(* Logix 5000 project; controller PRU vendor 1 type 14 code 107 rev 20.13; software revision 20.01; part 10 of 17 *)
(* tags used below, declared in another part *)
   AFI : BOOL;
   CR0_CON1_HTR1_GON : BOOL;   // ZONE 1 (L1,L2,L3)
   CR1_CON2_HTR2_GON : BOOL;   // ZONE 2 (L1,L2,L3)
   CR2_CON3_HTR3_GON : BOOL;   // ZONE 3 (L1,L2,L3)
   CR3_CON4_HTR4_GON : BOOL;   // ZONE 4 (L1) ZONE 5 (L2) ZONE 6 (L3)
   CR4_CON5_HTR5_GON : BOOL;   // ZONE 7 (L1) ZONE 8 (L2) ZONE 9 (L3)
   CYCLE_ION_DELAY1_TON : TIMER;
   CYCLE_ION_DELAY2_TON : TIMER;
   CYCLE_ION_DELAY3_TON : TIMER;
   CYCLE_ION_DELAY4_TON : TIMER;
   HEATERS_CYCLE_ION : BOOL;   // Heaters are commanded on.
   HTR1_CV : REAL;
   HTR1_MAX_CV_LIMIT : REAL;
   HTR1_POWER_CMD : REAL;
   HTR2_CV : REAL;
   HTR2_MAX_CV_LIMIT : DINT;
   HTR2_POWER_CMD : REAL;
   HTR3_CV : REAL;
   HTR3_MAX_CV_LIMIT : REAL;
   HTR3_POWER_CMD : REAL;
   HTR4_CV : REAL;
   HTR4_MAX_CV_LIMIT : REAL;
   HTR4_POWER_CMD : REAL;
   HTR5_CV : REAL;
   HTR5_MAX_CV_LIMIT : REAL;
   HTR5_POWER_CMD : REAL;
   HTR6_CV : REAL;
   HTR6_MAX_CV_LIMIT : REAL;
   HTR6_POWER_CMD : REAL;
   HTR7_CV : REAL;
   HTR7_MAX_CV_LIMIT : REAL;
   HTR7_POWER_CMD : REAL;
   HTR8_CV : REAL;
   HTR8_MAX_CV_LIMIT : REAL;
   HTR8_POWER_CMD : REAL;
   HTR9_CV : REAL;
   HTR9_MAX_CV_LIMIT : REAL;
   HTR9_POWER_CMD : REAL;
   PID_1_MODE_LOCAL : BOOL;
   PID_2_MODE_LOCAL : BOOL;
   PID_3_MODE_LOCAL : BOOL;
   PID_4_MODE_LOCAL : BOOL;
   PID_5_MODE_LOCAL : BOOL;
   PID_6_MODE_LOCAL : BOOL;
   PID_7_MODE_LOCAL : BOOL;
   PID_8_MODE_LOCAL : BOOL;
   PID_9_MODE_LOCAL : BOOL;
   PID_ZONE_1 : PID;
   PID_ZONE_1_MANUAL_SETPOINT : REAL;
   PID_ZONE_1_SETPOINT : DINT;
   PID_ZONE_2 : PID;
   PID_ZONE_2_MANUAL_SETPOINT : REAL;
   PID_ZONE_2_SETPOINT : DINT;
   PID_ZONE_3 : PID;
   PID_ZONE_3_MANUAL_SETPOINT : REAL;
   PID_ZONE_3_SETPOINT : DINT;
   PID_ZONE_4 : PID;
   PID_ZONE_4_MANUAL_SETPOINT : REAL;
   PID_ZONE_4_SETPOINT : DINT;
   PID_ZONE_5 : PID;
   PID_ZONE_5_MANUAL_SETPOINT : REAL;
   PID_ZONE_5_SETPOINT : REAL;
   PID_ZONE_6 : PID;
   PID_ZONE_6_MANUAL_SETPOINT : REAL;
   PID_ZONE_6_SETPOINT : REAL;
   PID_ZONE_7 : PID;
   PID_ZONE_7_MANUAL_SETPOINT : REAL;
   PID_ZONE_7_SETPOINT : DINT;
   PID_ZONE_8 : PID;
   PID_ZONE_8_MANUAL_SETPOINT : REAL;
   PID_ZONE_8_SETPOINT : DINT;
   PID_ZONE_9 : PID;
   PID_ZONE_9_MANUAL_SETPOINT : REAL;
   PID_ZONE_9_SETPOINT : DINT;
   STANDBY_MODE_ION : BOOL;
   STANDBY_TEMPERATURE_SETPOINT : REAL;
   TEMPERATURE_SETPOINT_IS_RAMPING : BOOL;
   TEST_HTR1_CV_LIMIT : BOOL;
   TEST_HTR2_CV_LIMIT : BOOL;
   TEST_HTR3_CV_LIMIT : BOOL;
   TEST_HTR4_CV_LIMIT : BOOL;
   TEST_HTR5_CV_LIMIT : BOOL;
   TEST_HTR6_CV_LIMIT : BOOL;
   TEST_HTR7_CV_LIMIT : BOOL;
   TEST_HTR8_CV_LIMIT : BOOL;
   TEST_HTR9_CV_LIMIT : BOOL;
   ZONE_1_TEMP_AVE : DINT;
   ZONE_2_TEMP_AVE : REAL;
   ZONE_3_TEMP_AVE : REAL;
   ZONE_4_TEMP_AVE : REAL;
   ZONE_5_TEMP_AVE : REAL;
   ZONE_6_TEMP_AVE : REAL;
   ZONE_7_TEMP_AVE : REAL;
   ZONE_8_TEMP_AVE : REAL;
   ZONE_9_TEMP_AVE : REAL;
(* MainProgram, continued *)

ROUTINE C02_HEATER_PID_CONTROL   (* ladder *)
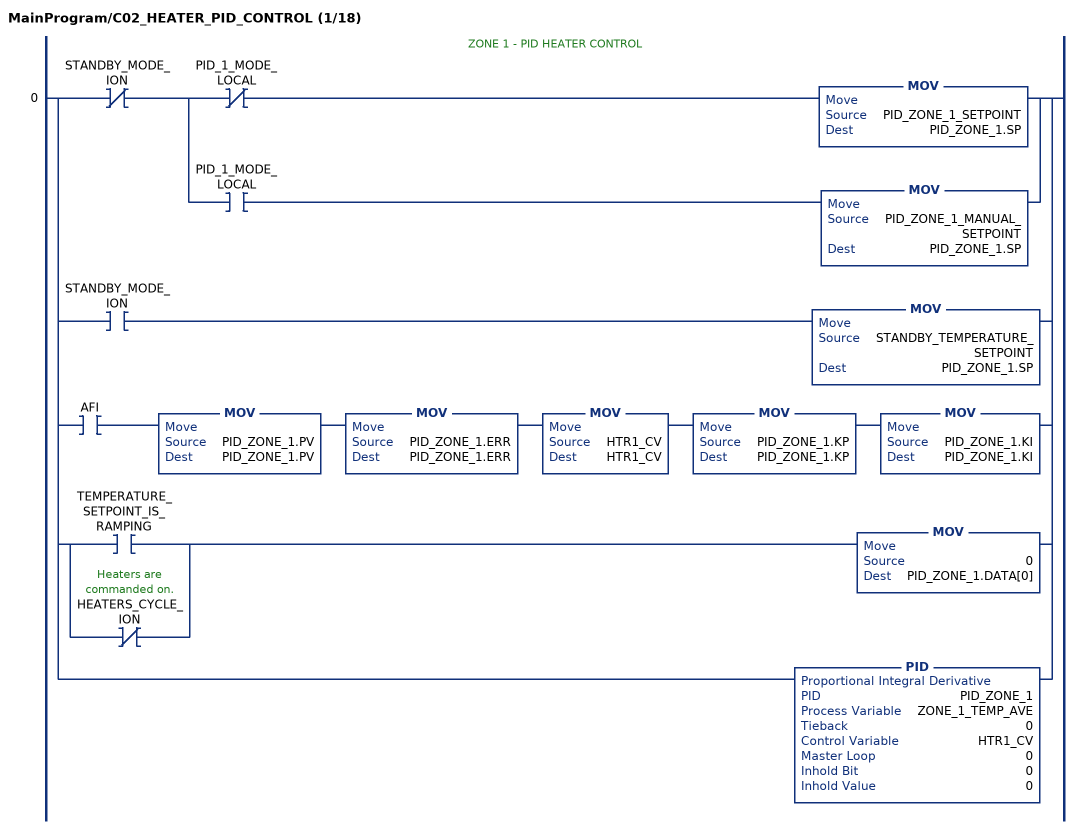
   // ZONE 1 - PID HEATER CONTROL
   0: [XIO(STANDBY_MODE_ION) [XIO(PID_1_MODE_LOCAL) MOV(PID_ZONE_1_SETPOINT,PID_ZONE_1.SP) ,XIC(PID_1_MODE_LOCAL) MOV(PID_ZONE_1_MANUAL_SETPOINT,PID_ZONE_1.SP) ] ,XIC(STANDBY_MODE_ION) MOV(STANDBY_TEMPERATURE_SETPOINT,PID_ZONE_1.SP) ,XIC(AFI) MOV(PID_ZONE_1.PV,PID_ZONE_1.PV) MOV(PID_ZONE_1.ERR,PID_ZONE_1.ERR) MOV(HTR1_CV,HTR1_CV) MOV(PID_ZONE_1.KP,PID_ZONE_1.KP) MOV(PID_ZONE_1.KI,PID_ZONE_1.KI) ,[XIC(TEMPERATURE_SETPOINT_IS_RAMPING) ,XIO(HEATERS_CYCLE_ION) ] MOV(0,PID_ZONE_1.DATA[0]) ,PID(PID_ZONE_1,ZONE_1_TEMP_AVE,0,HTR1_CV,0,0,0) ];
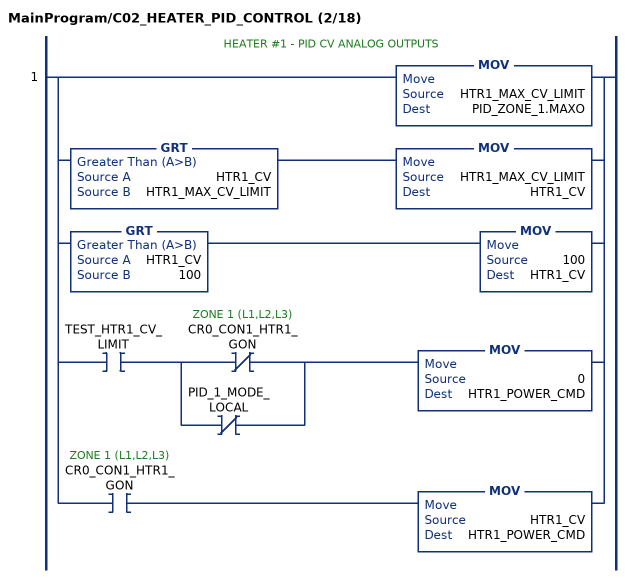
   // HEATER #1 - PID CV ANALOG OUTPUTS
   1: [MOV(HTR1_MAX_CV_LIMIT,PID_ZONE_1.MAXO) ,GRT(HTR1_CV,HTR1_MAX_CV_LIMIT) MOV(HTR1_MAX_CV_LIMIT,HTR1_CV) ,GRT(HTR1_CV,100) MOV(100,HTR1_CV) ,XIC(TEST_HTR1_CV_LIMIT) [XIO(CR0_CON1_HTR1_GON) ,XIO(PID_1_MODE_LOCAL) ] MOV(0,HTR1_POWER_CMD) ,XIC(CR0_CON1_HTR1_GON) MOV(HTR1_CV,HTR1_POWER_CMD) ];
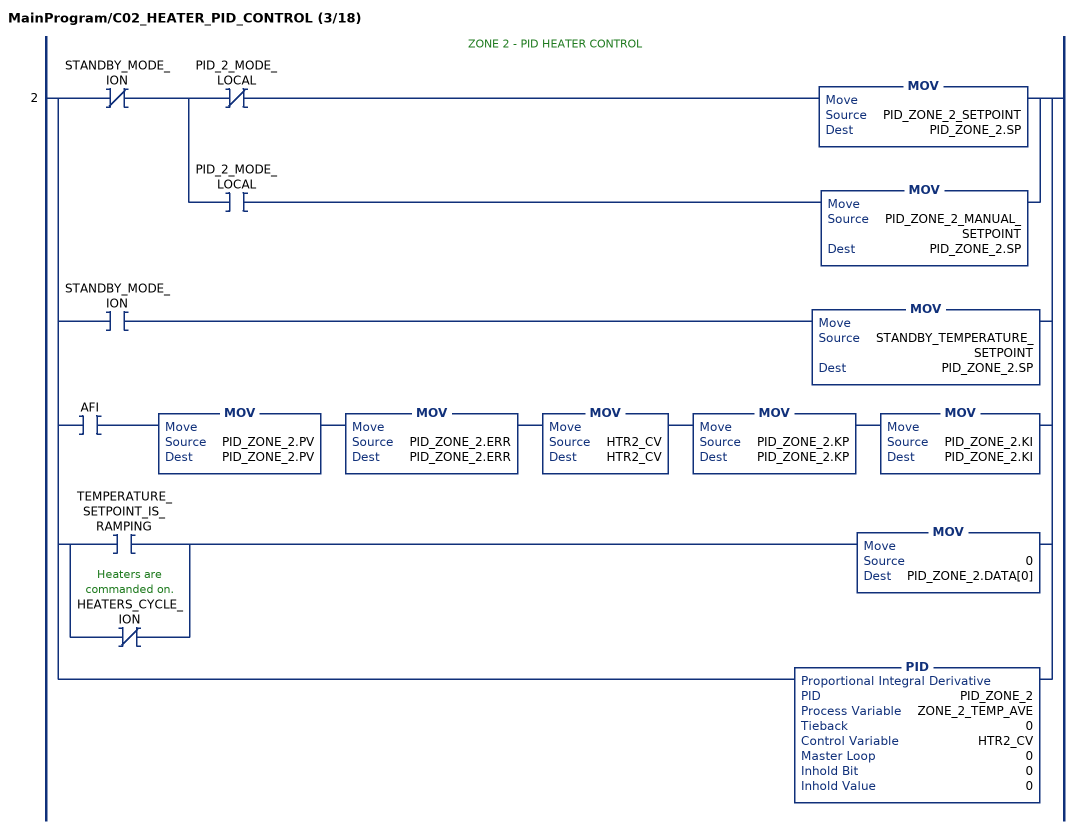
   // ZONE 2 - PID HEATER CONTROL
   2: [XIO(STANDBY_MODE_ION) [XIO(PID_2_MODE_LOCAL) MOV(PID_ZONE_2_SETPOINT,PID_ZONE_2.SP) ,XIC(PID_2_MODE_LOCAL) MOV(PID_ZONE_2_MANUAL_SETPOINT,PID_ZONE_2.SP) ] ,XIC(STANDBY_MODE_ION) MOV(STANDBY_TEMPERATURE_SETPOINT,PID_ZONE_2.SP) ,XIC(AFI) MOV(PID_ZONE_2.PV,PID_ZONE_2.PV) MOV(PID_ZONE_2.ERR,PID_ZONE_2.ERR) MOV(HTR2_CV,HTR2_CV) MOV(PID_ZONE_2.KP,PID_ZONE_2.KP) MOV(PID_ZONE_2.KI,PID_ZONE_2.KI) ,[XIC(TEMPERATURE_SETPOINT_IS_RAMPING) ,XIO(HEATERS_CYCLE_ION) ] MOV(0,PID_ZONE_2.DATA[0]) ,PID(PID_ZONE_2,ZONE_2_TEMP_AVE,0,HTR2_CV,0,0,0) ];
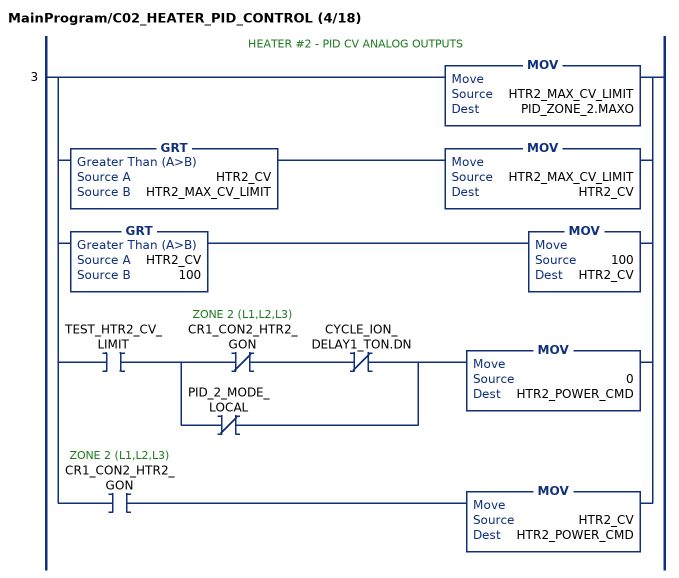
   // HEATER #2 - PID CV ANALOG OUTPUTS
   3: [MOV(HTR2_MAX_CV_LIMIT,PID_ZONE_2.MAXO) ,GRT(HTR2_CV,HTR2_MAX_CV_LIMIT) MOV(HTR2_MAX_CV_LIMIT,HTR2_CV) ,GRT(HTR2_CV,100) MOV(100,HTR2_CV) ,XIC(TEST_HTR2_CV_LIMIT) [XIO(CR1_CON2_HTR2_GON) XIO(CYCLE_ION_DELAY1_TON.DN) ,XIO(PID_2_MODE_LOCAL) ] MOV(0,HTR2_POWER_CMD) ,XIC(CR1_CON2_HTR2_GON) MOV(HTR2_CV,HTR2_POWER_CMD) ];
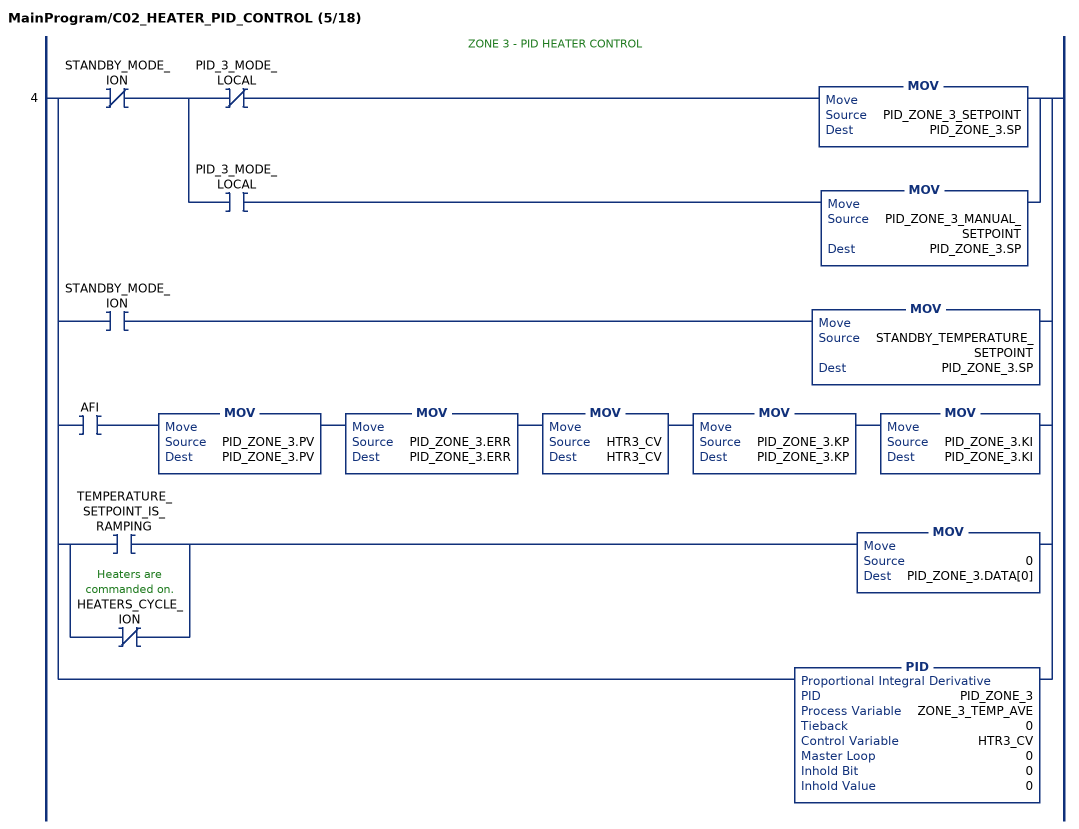
   // ZONE 3 - PID HEATER CONTROL
   4: [XIO(STANDBY_MODE_ION) [XIO(PID_3_MODE_LOCAL) MOV(PID_ZONE_3_SETPOINT,PID_ZONE_3.SP) ,XIC(PID_3_MODE_LOCAL) MOV(PID_ZONE_3_MANUAL_SETPOINT,PID_ZONE_3.SP) ] ,XIC(STANDBY_MODE_ION) MOV(STANDBY_TEMPERATURE_SETPOINT,PID_ZONE_3.SP) ,XIC(AFI) MOV(PID_ZONE_3.PV,PID_ZONE_3.PV) MOV(PID_ZONE_3.ERR,PID_ZONE_3.ERR) MOV(HTR3_CV,HTR3_CV) MOV(PID_ZONE_3.KP,PID_ZONE_3.KP) MOV(PID_ZONE_3.KI,PID_ZONE_3.KI) ,[XIC(TEMPERATURE_SETPOINT_IS_RAMPING) ,XIO(HEATERS_CYCLE_ION) ] MOV(0,PID_ZONE_3.DATA[0]) ,PID(PID_ZONE_3,ZONE_3_TEMP_AVE,0,HTR3_CV,0,0,0) ];
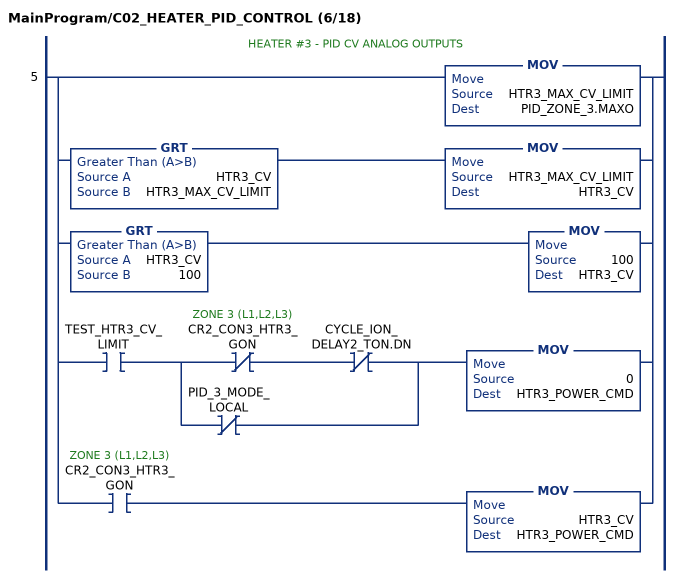
   // HEATER #3 - PID CV ANALOG OUTPUTS
   5: [MOV(HTR3_MAX_CV_LIMIT,PID_ZONE_3.MAXO) ,GRT(HTR3_CV,HTR3_MAX_CV_LIMIT) MOV(HTR3_MAX_CV_LIMIT,HTR3_CV) ,GRT(HTR3_CV,100) MOV(100,HTR3_CV) ,XIC(TEST_HTR3_CV_LIMIT) [XIO(CR2_CON3_HTR3_GON) XIO(CYCLE_ION_DELAY2_TON.DN) ,XIO(PID_3_MODE_LOCAL) ] MOV(0,HTR3_POWER_CMD) ,XIC(CR2_CON3_HTR3_GON) MOV(HTR3_CV,HTR3_POWER_CMD) ];
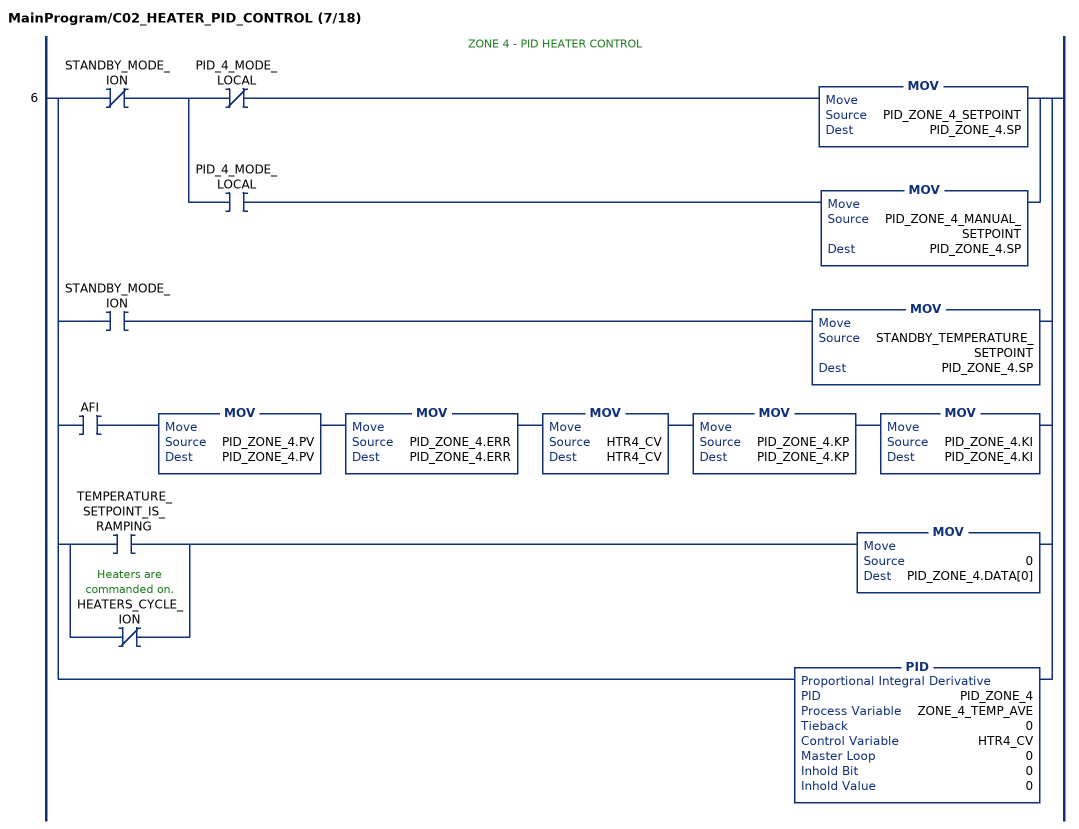
   // ZONE 4 - PID HEATER CONTROL
   6: [XIO(STANDBY_MODE_ION) [XIO(PID_4_MODE_LOCAL) MOV(PID_ZONE_4_SETPOINT,PID_ZONE_4.SP) ,XIC(PID_4_MODE_LOCAL) MOV(PID_ZONE_4_MANUAL_SETPOINT,PID_ZONE_4.SP) ] ,XIC(STANDBY_MODE_ION) MOV(STANDBY_TEMPERATURE_SETPOINT,PID_ZONE_4.SP) ,XIC(AFI) MOV(PID_ZONE_4.PV,PID_ZONE_4.PV) MOV(PID_ZONE_4.ERR,PID_ZONE_4.ERR) MOV(HTR4_CV,HTR4_CV) MOV(PID_ZONE_4.KP,PID_ZONE_4.KP) MOV(PID_ZONE_4.KI,PID_ZONE_4.KI) ,[XIC(TEMPERATURE_SETPOINT_IS_RAMPING) ,XIO(HEATERS_CYCLE_ION) ] MOV(0,PID_ZONE_4.DATA[0]) ,PID(PID_ZONE_4,ZONE_4_TEMP_AVE,0,HTR4_CV,0,0,0) ];
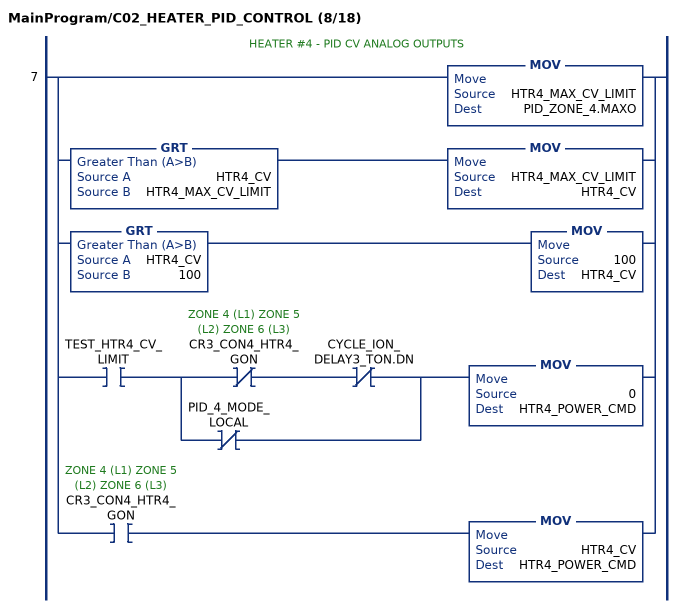
   // HEATER #4 - PID CV ANALOG OUTPUTS
   7: [MOV(HTR4_MAX_CV_LIMIT,PID_ZONE_4.MAXO) ,GRT(HTR4_CV,HTR4_MAX_CV_LIMIT) MOV(HTR4_MAX_CV_LIMIT,HTR4_CV) ,GRT(HTR4_CV,100) MOV(100,HTR4_CV) ,XIC(TEST_HTR4_CV_LIMIT) [XIO(CR3_CON4_HTR4_GON) XIO(CYCLE_ION_DELAY3_TON.DN) ,XIO(PID_4_MODE_LOCAL) ] MOV(0,HTR4_POWER_CMD) ,XIC(CR3_CON4_HTR4_GON) MOV(HTR4_CV,HTR4_POWER_CMD) ];
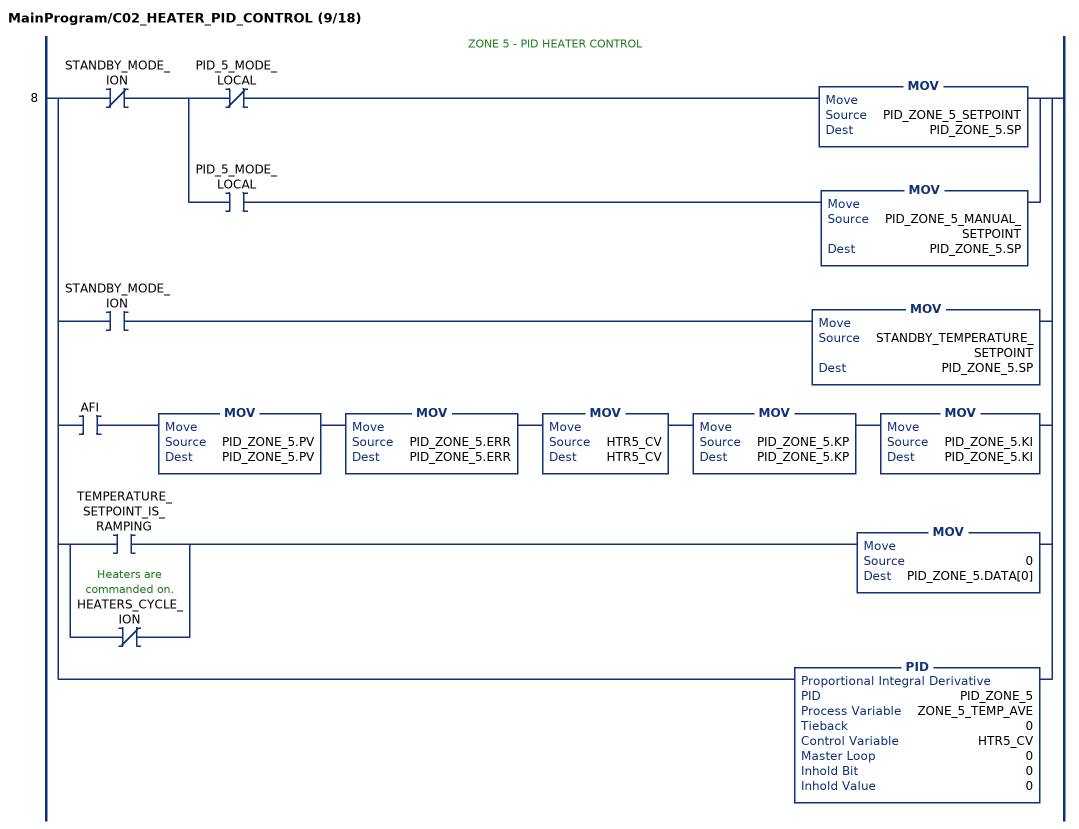
   // ZONE 5 - PID HEATER CONTROL
   8: [XIO(STANDBY_MODE_ION) [XIO(PID_5_MODE_LOCAL) MOV(PID_ZONE_5_SETPOINT,PID_ZONE_5.SP) ,XIC(PID_5_MODE_LOCAL) MOV(PID_ZONE_5_MANUAL_SETPOINT,PID_ZONE_5.SP) ] ,XIC(STANDBY_MODE_ION) MOV(STANDBY_TEMPERATURE_SETPOINT,PID_ZONE_5.SP) ,XIC(AFI) MOV(PID_ZONE_5.PV,PID_ZONE_5.PV) MOV(PID_ZONE_5.ERR,PID_ZONE_5.ERR) MOV(HTR5_CV,HTR5_CV) MOV(PID_ZONE_5.KP,PID_ZONE_5.KP) MOV(PID_ZONE_5.KI,PID_ZONE_5.KI) ,[XIC(TEMPERATURE_SETPOINT_IS_RAMPING) ,XIO(HEATERS_CYCLE_ION) ] MOV(0,PID_ZONE_5.DATA[0]) ,PID(PID_ZONE_5,ZONE_5_TEMP_AVE,0,HTR5_CV,0,0,0) ];
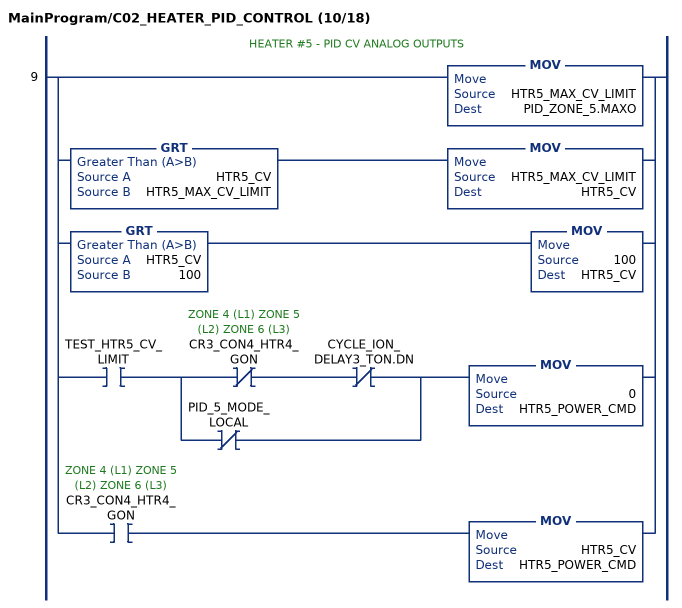
   // HEATER #5 - PID CV ANALOG OUTPUTS
   9: [MOV(HTR5_MAX_CV_LIMIT,PID_ZONE_5.MAXO) ,GRT(HTR5_CV,HTR5_MAX_CV_LIMIT) MOV(HTR5_MAX_CV_LIMIT,HTR5_CV) ,GRT(HTR5_CV,100) MOV(100,HTR5_CV) ,XIC(TEST_HTR5_CV_LIMIT) [XIO(CR3_CON4_HTR4_GON) XIO(CYCLE_ION_DELAY3_TON.DN) ,XIO(PID_5_MODE_LOCAL) ] MOV(0,HTR5_POWER_CMD) ,XIC(CR3_CON4_HTR4_GON) MOV(HTR5_CV,HTR5_POWER_CMD) ];
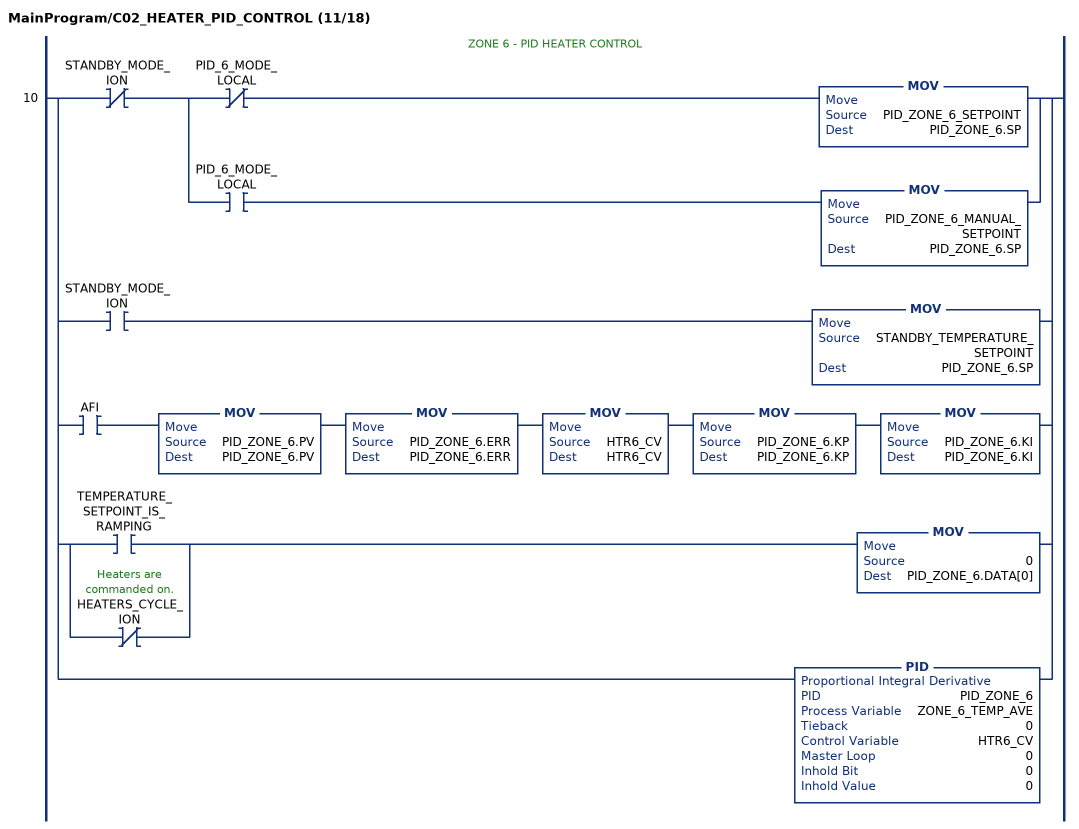
   // ZONE 6 - PID HEATER CONTROL
   10: [XIO(STANDBY_MODE_ION) [XIO(PID_6_MODE_LOCAL) MOV(PID_ZONE_6_SETPOINT,PID_ZONE_6.SP) ,XIC(PID_6_MODE_LOCAL) MOV(PID_ZONE_6_MANUAL_SETPOINT,PID_ZONE_6.SP) ] ,XIC(STANDBY_MODE_ION) MOV(STANDBY_TEMPERATURE_SETPOINT,PID_ZONE_6.SP) ,XIC(AFI) MOV(PID_ZONE_6.PV,PID_ZONE_6.PV) MOV(PID_ZONE_6.ERR,PID_ZONE_6.ERR) MOV(HTR6_CV,HTR6_CV) MOV(PID_ZONE_6.KP,PID_ZONE_6.KP) MOV(PID_ZONE_6.KI,PID_ZONE_6.KI) ,[XIC(TEMPERATURE_SETPOINT_IS_RAMPING) ,XIO(HEATERS_CYCLE_ION) ] MOV(0,PID_ZONE_6.DATA[0]) ,PID(PID_ZONE_6,ZONE_6_TEMP_AVE,0,HTR6_CV,0,0,0) ];
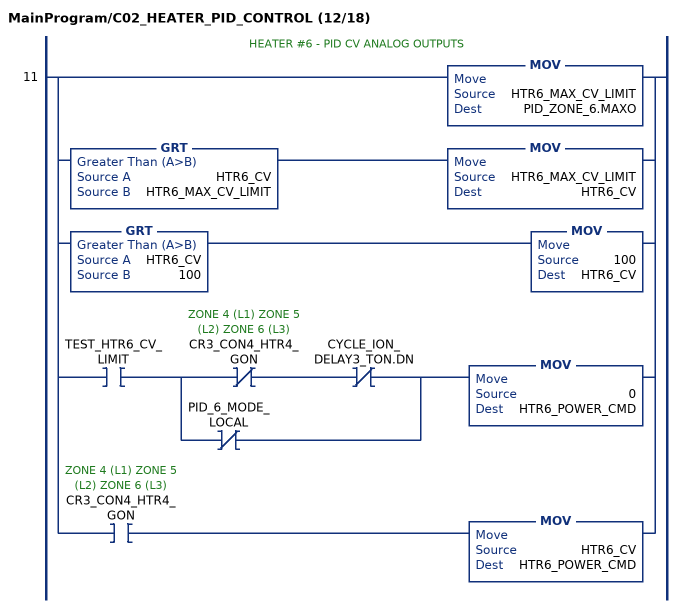
   // HEATER #6 - PID CV ANALOG OUTPUTS
   11: [MOV(HTR6_MAX_CV_LIMIT,PID_ZONE_6.MAXO) ,GRT(HTR6_CV,HTR6_MAX_CV_LIMIT) MOV(HTR6_MAX_CV_LIMIT,HTR6_CV) ,GRT(HTR6_CV,100) MOV(100,HTR6_CV) ,XIC(TEST_HTR6_CV_LIMIT) [XIO(CR3_CON4_HTR4_GON) XIO(CYCLE_ION_DELAY3_TON.DN) ,XIO(PID_6_MODE_LOCAL) ] MOV(0,HTR6_POWER_CMD) ,XIC(CR3_CON4_HTR4_GON) MOV(HTR6_CV,HTR6_POWER_CMD) ];
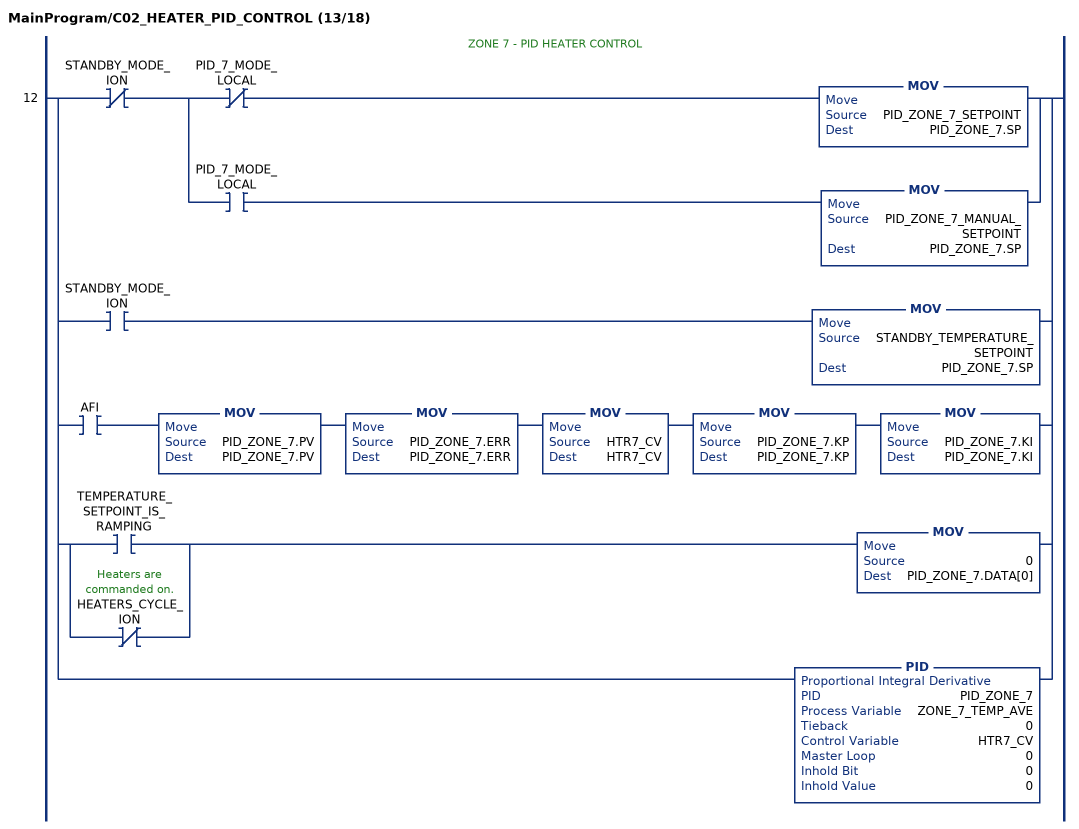
   // ZONE 7 - PID HEATER CONTROL
   12: [XIO(STANDBY_MODE_ION) [XIO(PID_7_MODE_LOCAL) MOV(PID_ZONE_7_SETPOINT,PID_ZONE_7.SP) ,XIC(PID_7_MODE_LOCAL) MOV(PID_ZONE_7_MANUAL_SETPOINT,PID_ZONE_7.SP) ] ,XIC(STANDBY_MODE_ION) MOV(STANDBY_TEMPERATURE_SETPOINT,PID_ZONE_7.SP) ,XIC(AFI) MOV(PID_ZONE_7.PV,PID_ZONE_7.PV) MOV(PID_ZONE_7.ERR,PID_ZONE_7.ERR) MOV(HTR7_CV,HTR7_CV) MOV(PID_ZONE_7.KP,PID_ZONE_7.KP) MOV(PID_ZONE_7.KI,PID_ZONE_7.KI) ,[XIC(TEMPERATURE_SETPOINT_IS_RAMPING) ,XIO(HEATERS_CYCLE_ION) ] MOV(0,PID_ZONE_7.DATA[0]) ,PID(PID_ZONE_7,ZONE_7_TEMP_AVE,0,HTR7_CV,0,0,0) ];
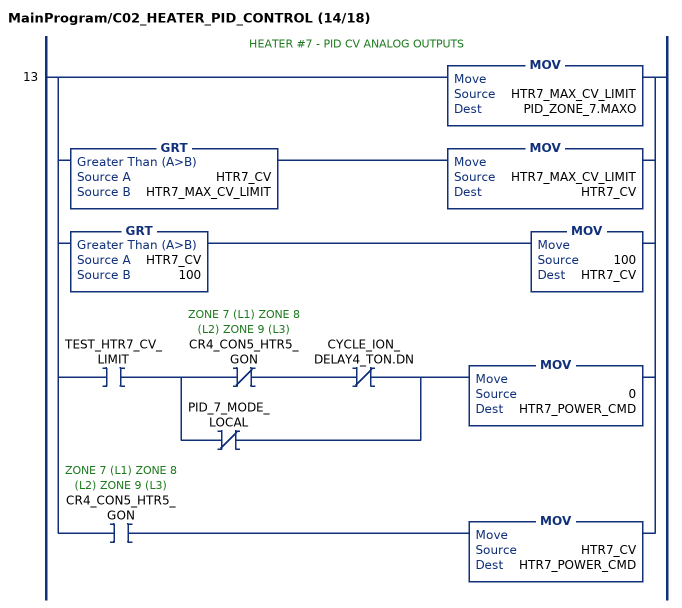
   // HEATER #7 - PID CV ANALOG OUTPUTS
   13: [MOV(HTR7_MAX_CV_LIMIT,PID_ZONE_7.MAXO) ,GRT(HTR7_CV,HTR7_MAX_CV_LIMIT) MOV(HTR7_MAX_CV_LIMIT,HTR7_CV) ,GRT(HTR7_CV,100) MOV(100,HTR7_CV) ,XIC(TEST_HTR7_CV_LIMIT) [XIO(CR4_CON5_HTR5_GON) XIO(CYCLE_ION_DELAY4_TON.DN) ,XIO(PID_7_MODE_LOCAL) ] MOV(0,HTR7_POWER_CMD) ,XIC(CR4_CON5_HTR5_GON) MOV(HTR7_CV,HTR7_POWER_CMD) ];
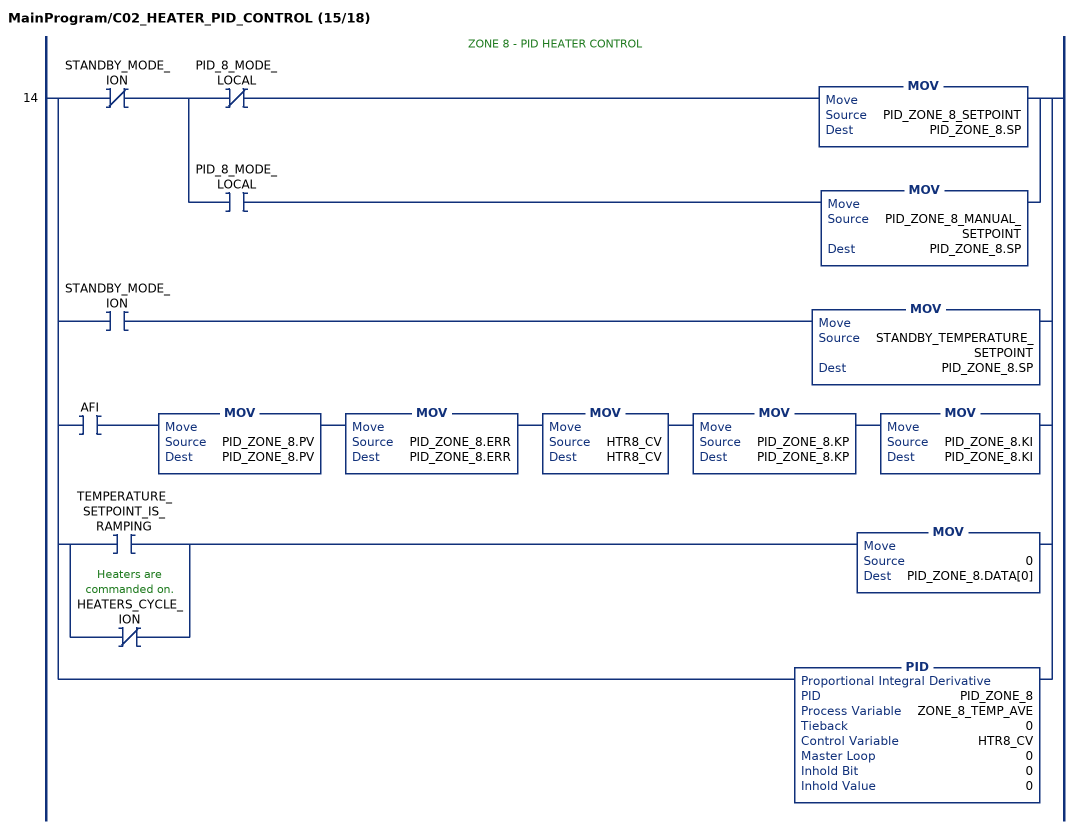
   // ZONE 8 - PID HEATER CONTROL
   14: [XIO(STANDBY_MODE_ION) [XIO(PID_8_MODE_LOCAL) MOV(PID_ZONE_8_SETPOINT,PID_ZONE_8.SP) ,XIC(PID_8_MODE_LOCAL) MOV(PID_ZONE_8_MANUAL_SETPOINT,PID_ZONE_8.SP) ] ,XIC(STANDBY_MODE_ION) MOV(STANDBY_TEMPERATURE_SETPOINT,PID_ZONE_8.SP) ,XIC(AFI) MOV(PID_ZONE_8.PV,PID_ZONE_8.PV) MOV(PID_ZONE_8.ERR,PID_ZONE_8.ERR) MOV(HTR8_CV,HTR8_CV) MOV(PID_ZONE_8.KP,PID_ZONE_8.KP) MOV(PID_ZONE_8.KI,PID_ZONE_8.KI) ,[XIC(TEMPERATURE_SETPOINT_IS_RAMPING) ,XIO(HEATERS_CYCLE_ION) ] MOV(0,PID_ZONE_8.DATA[0]) ,PID(PID_ZONE_8,ZONE_8_TEMP_AVE,0,HTR8_CV,0,0,0) ];
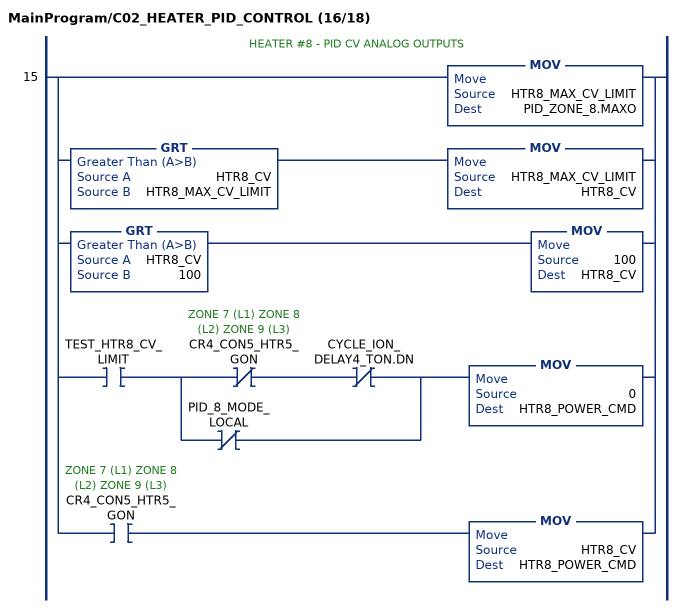
   // HEATER #8 - PID CV ANALOG OUTPUTS
   15: [MOV(HTR8_MAX_CV_LIMIT,PID_ZONE_8.MAXO) ,GRT(HTR8_CV,HTR8_MAX_CV_LIMIT) MOV(HTR8_MAX_CV_LIMIT,HTR8_CV) ,GRT(HTR8_CV,100) MOV(100,HTR8_CV) ,XIC(TEST_HTR8_CV_LIMIT) [XIO(CR4_CON5_HTR5_GON) XIO(CYCLE_ION_DELAY4_TON.DN) ,XIO(PID_8_MODE_LOCAL) ] MOV(0,HTR8_POWER_CMD) ,XIC(CR4_CON5_HTR5_GON) MOV(HTR8_CV,HTR8_POWER_CMD) ];
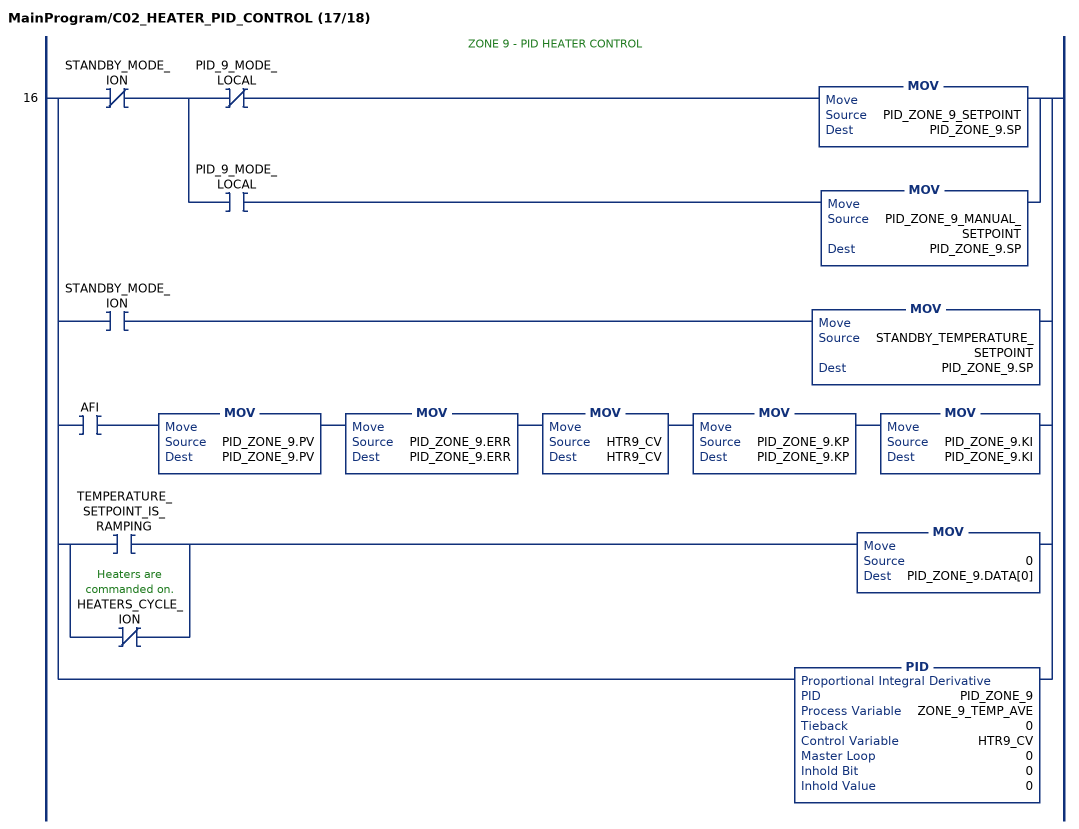
   // ZONE 9 - PID HEATER CONTROL
   16: [XIO(STANDBY_MODE_ION) [XIO(PID_9_MODE_LOCAL) MOV(PID_ZONE_9_SETPOINT,PID_ZONE_9.SP) ,XIC(PID_9_MODE_LOCAL) MOV(PID_ZONE_9_MANUAL_SETPOINT,PID_ZONE_9.SP) ] ,XIC(STANDBY_MODE_ION) MOV(STANDBY_TEMPERATURE_SETPOINT,PID_ZONE_9.SP) ,XIC(AFI) MOV(PID_ZONE_9.PV,PID_ZONE_9.PV) MOV(PID_ZONE_9.ERR,PID_ZONE_9.ERR) MOV(HTR9_CV,HTR9_CV) MOV(PID_ZONE_9.KP,PID_ZONE_9.KP) MOV(PID_ZONE_9.KI,PID_ZONE_9.KI) ,[XIC(TEMPERATURE_SETPOINT_IS_RAMPING) ,XIO(HEATERS_CYCLE_ION) ] MOV(0,PID_ZONE_9.DATA[0]) ,PID(PID_ZONE_9,ZONE_9_TEMP_AVE,0,HTR9_CV,0,0,0) ];
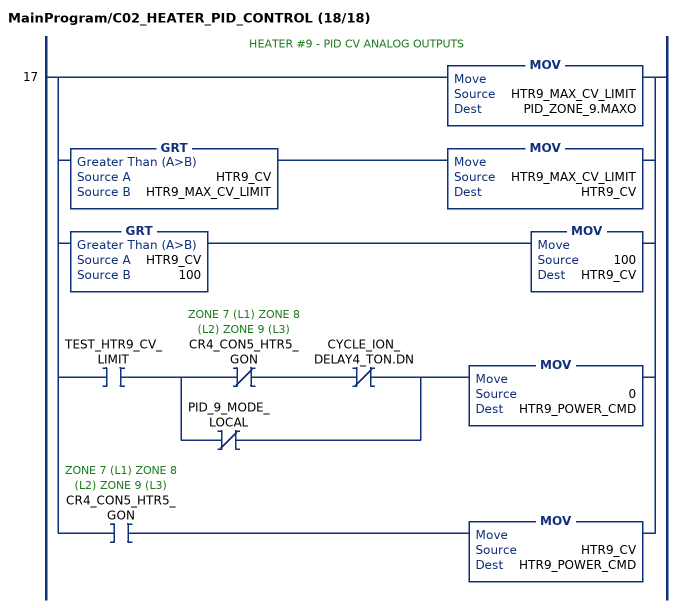
   // HEATER #9 - PID CV ANALOG OUTPUTS
   17: [MOV(HTR9_MAX_CV_LIMIT,PID_ZONE_9.MAXO) ,GRT(HTR9_CV,HTR9_MAX_CV_LIMIT) MOV(HTR9_MAX_CV_LIMIT,HTR9_CV) ,GRT(HTR9_CV,100) MOV(100,HTR9_CV) ,XIC(TEST_HTR9_CV_LIMIT) [XIO(CR4_CON5_HTR5_GON) XIO(CYCLE_ION_DELAY4_TON.DN) ,XIO(PID_9_MODE_LOCAL) ] MOV(0,HTR9_POWER_CMD) ,XIC(CR4_CON5_HTR5_GON) MOV(HTR9_CV,HTR9_POWER_CMD) ];
END_ROUTINE
